// ============================================
// DB_RecipeProgram1 - SpinningCam Program
// Lines: 445
// Generated by SpinningCam
// ============================================

DATA_BLOCK "DB_RecipeProgram1"
{ S7_Optimized_Access := 'TRUE' }
VERSION : 0.1
NON_RETAIN
    VAR
        Header : "RecipeHeader";
        Lines : Array[0..999] of "RecipeLine";
    END_VAR
BEGIN
    // Header
    Header.Name := 'SpinningCam Program';
    Header.LineCount := 445;
    Header.Valid := TRUE;
    Header.PreScanned := FALSE;
    Header.MinX := 0.000;
    Header.MaxX := 118.345;
    Header.MinZ := -188.810;
    Header.MaxZ := 0.000;

    // Recipe Lines (445 total)
    Lines[0].X := 0.000; Lines[0].Z := 0.000; Lines[0].F := 0; Lines[0].CMD := 0; Lines[0].Param := 0; // G0 Rapid
    Lines[1].X := 0.000; Lines[1].Z := 0.000; Lines[1].F := 0; Lines[1].CMD := 0; Lines[1].Param := 0; // G0 Rapid
    Lines[2].X := 0.000; Lines[2].Z := 0.000; Lines[2].F := 0; Lines[2].CMD := 10; Lines[2].Param := 101; // Tool Change T101
    Lines[3].X := 0.000; Lines[3].Z := 0.000; Lines[3].F := 0; Lines[3].CMD := 20; Lines[3].Param := 20; // Spindle ON 200 RPM
    Lines[4].X := 34.600; Lines[4].Z := -28.936; Lines[4].F := 0; Lines[4].CMD := 0; Lines[4].Param := 0; // G0 Rapid
    Lines[5].X := 35.427; Lines[5].Z := -29.545; Lines[5].F := 300; Lines[5].CMD := 1; Lines[5].Param := 0; // G1 Linear
    Lines[6].X := 36.268; Lines[6].Z := -30.173; Lines[6].F := 300; Lines[6].CMD := 1; Lines[6].Param := 0; // G1 Linear
    Lines[7].X := 37.121; Lines[7].Z := -30.818; Lines[7].F := 300; Lines[7].CMD := 1; Lines[7].Param := 0; // G1 Linear
    Lines[8].X := 37.986; Lines[8].Z := -31.481; Lines[8].F := 300; Lines[8].CMD := 1; Lines[8].Param := 0; // G1 Linear
    Lines[9].X := 38.860; Lines[9].Z := -32.160; Lines[9].F := 300; Lines[9].CMD := 1; Lines[9].Param := 0; // G1 Linear
    Lines[10].X := 39.744; Lines[10].Z := -32.855; Lines[10].F := 300; Lines[10].CMD := 1; Lines[10].Param := 0; // G1 Linear
    Lines[11].X := 40.636; Lines[11].Z := -33.566; Lines[11].F := 300; Lines[11].CMD := 1; Lines[11].Param := 0; // G1 Linear
    Lines[12].X := 41.535; Lines[12].Z := -34.291; Lines[12].F := 300; Lines[12].CMD := 1; Lines[12].Param := 0; // G1 Linear
    Lines[13].X := 42.441; Lines[13].Z := -35.031; Lines[13].F := 300; Lines[13].CMD := 1; Lines[13].Param := 0; // G1 Linear
    Lines[14].X := 43.351; Lines[14].Z := -35.785; Lines[14].F := 300; Lines[14].CMD := 1; Lines[14].Param := 0; // G1 Linear
    Lines[15].X := 44.265; Lines[15].Z := -36.552; Lines[15].F := 300; Lines[15].CMD := 1; Lines[15].Param := 0; // G1 Linear
    Lines[16].X := 45.183; Lines[16].Z := -37.332; Lines[16].F := 300; Lines[16].CMD := 1; Lines[16].Param := 0; // G1 Linear
    Lines[17].X := 46.102; Lines[17].Z := -38.124; Lines[17].F := 300; Lines[17].CMD := 1; Lines[17].Param := 0; // G1 Linear
    Lines[18].X := 47.022; Lines[18].Z := -38.928; Lines[18].F := 300; Lines[18].CMD := 1; Lines[18].Param := 0; // G1 Linear
    Lines[19].X := 47.942; Lines[19].Z := -39.743; Lines[19].F := 300; Lines[19].CMD := 1; Lines[19].Param := 0; // G1 Linear
    Lines[20].X := 48.861; Lines[20].Z := -40.568; Lines[20].F := 300; Lines[20].CMD := 1; Lines[20].Param := 0; // G1 Linear
    Lines[21].X := 49.777; Lines[21].Z := -41.404; Lines[21].F := 300; Lines[21].CMD := 1; Lines[21].Param := 0; // G1 Linear
    Lines[22].X := 50.691; Lines[22].Z := -42.249; Lines[22].F := 300; Lines[22].CMD := 1; Lines[22].Param := 0; // G1 Linear
    Lines[23].X := 51.600; Lines[23].Z := -43.103; Lines[23].F := 300; Lines[23].CMD := 1; Lines[23].Param := 0; // G1 Linear
    Lines[24].X := 52.503; Lines[24].Z := -43.965; Lines[24].F := 300; Lines[24].CMD := 1; Lines[24].Param := 0; // G1 Linear
    Lines[25].X := 53.401; Lines[25].Z := -44.835; Lines[25].F := 300; Lines[25].CMD := 1; Lines[25].Param := 0; // G1 Linear
    Lines[26].X := 54.291; Lines[26].Z := -45.713; Lines[26].F := 300; Lines[26].CMD := 1; Lines[26].Param := 0; // G1 Linear
    Lines[27].X := 55.172; Lines[27].Z := -46.597; Lines[27].F := 300; Lines[27].CMD := 1; Lines[27].Param := 0; // G1 Linear
    Lines[28].X := 56.044; Lines[28].Z := -47.488; Lines[28].F := 300; Lines[28].CMD := 1; Lines[28].Param := 0; // G1 Linear
    Lines[29].X := 56.905; Lines[29].Z := -48.384; Lines[29].F := 300; Lines[29].CMD := 1; Lines[29].Param := 0; // G1 Linear
    Lines[30].X := 57.755; Lines[30].Z := -49.285; Lines[30].F := 300; Lines[30].CMD := 1; Lines[30].Param := 0; // G1 Linear
    Lines[31].X := 58.592; Lines[31].Z := -50.191; Lines[31].F := 300; Lines[31].CMD := 1; Lines[31].Param := 0; // G1 Linear
    Lines[32].X := 59.415; Lines[32].Z := -51.101; Lines[32].F := 300; Lines[32].CMD := 1; Lines[32].Param := 0; // G1 Linear
    Lines[33].X := 60.224; Lines[33].Z := -52.014; Lines[33].F := 300; Lines[33].CMD := 1; Lines[33].Param := 0; // G1 Linear
    Lines[34].X := 61.017; Lines[34].Z := -52.931; Lines[34].F := 300; Lines[34].CMD := 1; Lines[34].Param := 0; // G1 Linear
    Lines[35].X := 61.793; Lines[35].Z := -53.849; Lines[35].F := 300; Lines[35].CMD := 1; Lines[35].Param := 0; // G1 Linear
    Lines[36].X := 62.551; Lines[36].Z := -54.770; Lines[36].F := 300; Lines[36].CMD := 1; Lines[36].Param := 0; // G1 Linear
    Lines[37].X := 63.291; Lines[37].Z := -55.692; Lines[37].F := 300; Lines[37].CMD := 1; Lines[37].Param := 0; // G1 Linear
    Lines[38].X := 64.010; Lines[38].Z := -56.614; Lines[38].F := 300; Lines[38].CMD := 1; Lines[38].Param := 0; // G1 Linear
    Lines[39].X := 64.709; Lines[39].Z := -57.537; Lines[39].F := 300; Lines[39].CMD := 1; Lines[39].Param := 0; // G1 Linear
    Lines[40].X := 65.385; Lines[40].Z := -58.460; Lines[40].F := 300; Lines[40].CMD := 1; Lines[40].Param := 0; // G1 Linear
    Lines[41].X := 66.039; Lines[41].Z := -59.381; Lines[41].F := 300; Lines[41].CMD := 1; Lines[41].Param := 0; // G1 Linear
    Lines[42].X := 66.668; Lines[42].Z := -60.301; Lines[42].F := 300; Lines[42].CMD := 1; Lines[42].Param := 0; // G1 Linear
    Lines[43].X := 67.273; Lines[43].Z := -61.220; Lines[43].F := 300; Lines[43].CMD := 1; Lines[43].Param := 0; // G1 Linear
    Lines[44].X := 67.851; Lines[44].Z := -62.135; Lines[44].F := 300; Lines[44].CMD := 1; Lines[44].Param := 0; // G1 Linear
    Lines[45].X := 68.402; Lines[45].Z := -63.048; Lines[45].F := 300; Lines[45].CMD := 1; Lines[45].Param := 0; // G1 Linear
    Lines[46].X := 68.924; Lines[46].Z := -63.957; Lines[46].F := 300; Lines[46].CMD := 1; Lines[46].Param := 0; // G1 Linear
    Lines[47].X := 69.418; Lines[47].Z := -64.862; Lines[47].F := 300; Lines[47].CMD := 1; Lines[47].Param := 0; // G1 Linear
    Lines[48].X := 69.881; Lines[48].Z := -65.762; Lines[48].F := 300; Lines[48].CMD := 1; Lines[48].Param := 0; // G1 Linear
    Lines[49].X := 70.313; Lines[49].Z := -66.657; Lines[49].F := 300; Lines[49].CMD := 1; Lines[49].Param := 0; // G1 Linear
    Lines[50].X := 70.712; Lines[50].Z := -67.546; Lines[50].F := 300; Lines[50].CMD := 1; Lines[50].Param := 0; // G1 Linear
    Lines[51].X := 71.078; Lines[51].Z := -68.428; Lines[51].F := 300; Lines[51].CMD := 1; Lines[51].Param := 0; // G1 Linear
    Lines[52].X := 71.409; Lines[52].Z := -69.304; Lines[52].F := 300; Lines[52].CMD := 1; Lines[52].Param := 0; // G1 Linear
    Lines[53].X := 71.705; Lines[53].Z := -70.173; Lines[53].F := 300; Lines[53].CMD := 1; Lines[53].Param := 0; // G1 Linear
    Lines[54].X := 71.964; Lines[54].Z := -71.033; Lines[54].F := 300; Lines[54].CMD := 1; Lines[54].Param := 0; // G1 Linear
    Lines[55].X := 72.186; Lines[55].Z := -71.885; Lines[55].F := 300; Lines[55].CMD := 1; Lines[55].Param := 0; // G1 Linear
    Lines[56].X := 72.369; Lines[56].Z := -72.728; Lines[56].F := 300; Lines[56].CMD := 1; Lines[56].Param := 0; // G1 Linear
    Lines[57].X := 72.512; Lines[57].Z := -73.561; Lines[57].F := 300; Lines[57].CMD := 1; Lines[57].Param := 0; // G1 Linear
    Lines[58].X := 72.614; Lines[58].Z := -74.384; Lines[58].F := 300; Lines[58].CMD := 1; Lines[58].Param := 0; // G1 Linear
    Lines[59].X := 72.675; Lines[59].Z := -75.196; Lines[59].F := 300; Lines[59].CMD := 1; Lines[59].Param := 0; // G1 Linear
    Lines[60].X := 72.693; Lines[60].Z := -75.997; Lines[60].F := 300; Lines[60].CMD := 1; Lines[60].Param := 0; // G1 Linear
    Lines[61].X := 72.667; Lines[61].Z := -76.786; Lines[61].F := 300; Lines[61].CMD := 1; Lines[61].Param := 0; // G1 Linear
    Lines[62].X := 72.596; Lines[62].Z := -77.563; Lines[62].F := 300; Lines[62].CMD := 1; Lines[62].Param := 0; // G1 Linear
    Lines[63].X := 72.480; Lines[63].Z := -78.327; Lines[63].F := 300; Lines[63].CMD := 1; Lines[63].Param := 0; // G1 Linear
    Lines[64].X := 72.316; Lines[64].Z := -79.078; Lines[64].F := 300; Lines[64].CMD := 1; Lines[64].Param := 0; // G1 Linear
    Lines[65].X := 72.104; Lines[65].Z := -79.814; Lines[65].F := 300; Lines[65].CMD := 1; Lines[65].Param := 0; // G1 Linear
    Lines[66].X := 71.843; Lines[66].Z := -80.536; Lines[66].F := 300; Lines[66].CMD := 1; Lines[66].Param := 0; // G1 Linear
    Lines[67].X := 71.532; Lines[67].Z := -81.243; Lines[67].F := 300; Lines[67].CMD := 1; Lines[67].Param := 0; // G1 Linear
    Lines[68].X := 71.171; Lines[68].Z := -81.935; Lines[68].F := 300; Lines[68].CMD := 1; Lines[68].Param := 0; // G1 Linear
    Lines[69].X := 70.760; Lines[69].Z := -82.610; Lines[69].F := 300; Lines[69].CMD := 1; Lines[69].Param := 0; // G1 Linear
    Lines[70].X := 70.301; Lines[70].Z := -83.271; Lines[70].F := 300; Lines[70].CMD := 1; Lines[70].Param := 0; // G1 Linear
    Lines[71].X := 69.795; Lines[71].Z := -83.916; Lines[71].F := 300; Lines[71].CMD := 1; Lines[71].Param := 0; // G1 Linear
    Lines[72].X := 69.245; Lines[72].Z := -84.547; Lines[72].F := 300; Lines[72].CMD := 1; Lines[72].Param := 0; // G1 Linear
    Lines[73].X := 68.652; Lines[73].Z := -85.162; Lines[73].F := 300; Lines[73].CMD := 1; Lines[73].Param := 0; // G1 Linear
    Lines[74].X := 68.018; Lines[74].Z := -85.762; Lines[74].F := 300; Lines[74].CMD := 1; Lines[74].Param := 0; // G1 Linear
    Lines[75].X := 67.344; Lines[75].Z := -86.348; Lines[75].F := 300; Lines[75].CMD := 1; Lines[75].Param := 0; // G1 Linear
    Lines[76].X := 66.632; Lines[76].Z := -86.919; Lines[76].F := 300; Lines[76].CMD := 1; Lines[76].Param := 0; // G1 Linear
    Lines[77].X := 65.884; Lines[77].Z := -87.476; Lines[77].F := 300; Lines[77].CMD := 1; Lines[77].Param := 0; // G1 Linear
    Lines[78].X := 65.101; Lines[78].Z := -88.019; Lines[78].F := 300; Lines[78].CMD := 1; Lines[78].Param := 0; // G1 Linear
    Lines[79].X := 64.284; Lines[79].Z := -88.547; Lines[79].F := 300; Lines[79].CMD := 1; Lines[79].Param := 0; // G1 Linear
    Lines[80].X := 63.436; Lines[80].Z := -89.062; Lines[80].F := 300; Lines[80].CMD := 1; Lines[80].Param := 0; // G1 Linear
    Lines[81].X := 62.558; Lines[81].Z := -89.562; Lines[81].F := 300; Lines[81].CMD := 1; Lines[81].Param := 0; // G1 Linear
    Lines[82].X := 61.652; Lines[82].Z := -90.049; Lines[82].F := 300; Lines[82].CMD := 1; Lines[82].Param := 0; // G1 Linear
    Lines[83].X := 60.719; Lines[83].Z := -90.523; Lines[83].F := 300; Lines[83].CMD := 1; Lines[83].Param := 0; // G1 Linear
    Lines[84].X := 59.761; Lines[84].Z := -90.982; Lines[84].F := 300; Lines[84].CMD := 1; Lines[84].Param := 0; // G1 Linear
    Lines[85].X := 58.780; Lines[85].Z := -91.429; Lines[85].F := 300; Lines[85].CMD := 1; Lines[85].Param := 0; // G1 Linear
    Lines[86].X := 57.777; Lines[86].Z := -91.862; Lines[86].F := 300; Lines[86].CMD := 1; Lines[86].Param := 0; // G1 Linear
    Lines[87].X := 56.754; Lines[87].Z := -92.283; Lines[87].F := 300; Lines[87].CMD := 1; Lines[87].Param := 0; // G1 Linear
    Lines[88].X := 55.712; Lines[88].Z := -92.690; Lines[88].F := 300; Lines[88].CMD := 1; Lines[88].Param := 0; // G1 Linear
    Lines[89].X := 54.654; Lines[89].Z := -93.085; Lines[89].F := 300; Lines[89].CMD := 1; Lines[89].Param := 0; // G1 Linear
    Lines[90].X := 53.580; Lines[90].Z := -93.467; Lines[90].F := 300; Lines[90].CMD := 1; Lines[90].Param := 0; // G1 Linear
    Lines[91].X := 52.493; Lines[91].Z := -93.836; Lines[91].F := 300; Lines[91].CMD := 1; Lines[91].Param := 0; // G1 Linear
    Lines[92].X := 51.393; Lines[92].Z := -94.193; Lines[92].F := 300; Lines[92].CMD := 1; Lines[92].Param := 0; // G1 Linear
    Lines[93].X := 50.284; Lines[93].Z := -94.538; Lines[93].F := 300; Lines[93].CMD := 1; Lines[93].Param := 0; // G1 Linear
    Lines[94].X := 49.165; Lines[94].Z := -94.871; Lines[94].F := 300; Lines[94].CMD := 1; Lines[94].Param := 0; // G1 Linear
    Lines[95].X := 48.040; Lines[95].Z := -95.192; Lines[95].F := 300; Lines[95].CMD := 1; Lines[95].Param := 0; // G1 Linear
    Lines[96].X := 46.909; Lines[96].Z := -95.501; Lines[96].F := 300; Lines[96].CMD := 1; Lines[96].Param := 0; // G1 Linear
    Lines[97].X := 45.775; Lines[97].Z := -95.798; Lines[97].F := 300; Lines[97].CMD := 1; Lines[97].Param := 0; // G1 Linear
    Lines[98].X := 44.638; Lines[98].Z := -96.084; Lines[98].F := 300; Lines[98].CMD := 1; Lines[98].Param := 0; // G1 Linear
    Lines[99].X := 43.501; Lines[99].Z := -96.358; Lines[99].F := 300; Lines[99].CMD := 1; Lines[99].Param := 0; // G1 Linear
    Lines[100].X := 42.364; Lines[100].Z := -96.621; Lines[100].F := 300; Lines[100].CMD := 1; Lines[100].Param := 0; // G1 Linear
    Lines[101].X := 41.231; Lines[101].Z := -96.873; Lines[101].F := 300; Lines[101].CMD := 1; Lines[101].Param := 0; // G1 Linear
    Lines[102].X := 40.102; Lines[102].Z := -97.114; Lines[102].F := 300; Lines[102].CMD := 1; Lines[102].Param := 0; // G1 Linear
    Lines[103].X := 38.979; Lines[103].Z := -97.344; Lines[103].F := 300; Lines[103].CMD := 1; Lines[103].Param := 0; // G1 Linear
    Lines[104].X := 37.863; Lines[104].Z := -97.564; Lines[104].F := 300; Lines[104].CMD := 1; Lines[104].Param := 0; // G1 Linear
    Lines[105].X := 36.757; Lines[105].Z := -97.772; Lines[105].F := 300; Lines[105].CMD := 1; Lines[105].Param := 0; // G1 Linear
    Lines[106].X := 35.662; Lines[106].Z := -97.971; Lines[106].F := 300; Lines[106].CMD := 1; Lines[106].Param := 0; // G1 Linear
    Lines[107].X := 34.579; Lines[107].Z := -98.159; Lines[107].F := 300; Lines[107].CMD := 1; Lines[107].Param := 0; // G1 Linear
    Lines[108].X := 33.511; Lines[108].Z := -98.337; Lines[108].F := 300; Lines[108].CMD := 1; Lines[108].Param := 0; // G1 Linear
    Lines[109].X := 32.458; Lines[109].Z := -98.504; Lines[109].F := 300; Lines[109].CMD := 1; Lines[109].Param := 0; // G1 Linear
    Lines[110].X := 31.422; Lines[110].Z := -98.662; Lines[110].F := 300; Lines[110].CMD := 1; Lines[110].Param := 0; // G1 Linear
    Lines[111].X := 30.406; Lines[111].Z := -98.810; Lines[111].F := 300; Lines[111].CMD := 1; Lines[111].Param := 0; // G1 Linear
    Lines[112].X := 10.406; Lines[112].Z := -78.810; Lines[112].F := 0; Lines[112].CMD := 0; Lines[112].Param := 0; // G0 Rapid
    Lines[113].X := 49.600; Lines[113].Z := -58.936; Lines[113].F := 0; Lines[113].CMD := 0; Lines[113].Param := 0; // G0 Rapid
    Lines[114].X := 50.427; Lines[114].Z := -59.545; Lines[114].F := 300; Lines[114].CMD := 1; Lines[114].Param := 0; // G1 Linear
    Lines[115].X := 51.268; Lines[115].Z := -60.173; Lines[115].F := 300; Lines[115].CMD := 1; Lines[115].Param := 0; // G1 Linear
    Lines[116].X := 52.121; Lines[116].Z := -60.818; Lines[116].F := 300; Lines[116].CMD := 1; Lines[116].Param := 0; // G1 Linear
    Lines[117].X := 52.986; Lines[117].Z := -61.481; Lines[117].F := 300; Lines[117].CMD := 1; Lines[117].Param := 0; // G1 Linear
    Lines[118].X := 53.860; Lines[118].Z := -62.160; Lines[118].F := 300; Lines[118].CMD := 1; Lines[118].Param := 0; // G1 Linear
    Lines[119].X := 54.744; Lines[119].Z := -62.855; Lines[119].F := 300; Lines[119].CMD := 1; Lines[119].Param := 0; // G1 Linear
    Lines[120].X := 55.636; Lines[120].Z := -63.566; Lines[120].F := 300; Lines[120].CMD := 1; Lines[120].Param := 0; // G1 Linear
    Lines[121].X := 56.535; Lines[121].Z := -64.291; Lines[121].F := 300; Lines[121].CMD := 1; Lines[121].Param := 0; // G1 Linear
    Lines[122].X := 57.441; Lines[122].Z := -65.031; Lines[122].F := 300; Lines[122].CMD := 1; Lines[122].Param := 0; // G1 Linear
    Lines[123].X := 58.351; Lines[123].Z := -65.785; Lines[123].F := 300; Lines[123].CMD := 1; Lines[123].Param := 0; // G1 Linear
    Lines[124].X := 59.265; Lines[124].Z := -66.552; Lines[124].F := 300; Lines[124].CMD := 1; Lines[124].Param := 0; // G1 Linear
    Lines[125].X := 60.183; Lines[125].Z := -67.332; Lines[125].F := 300; Lines[125].CMD := 1; Lines[125].Param := 0; // G1 Linear
    Lines[126].X := 61.102; Lines[126].Z := -68.124; Lines[126].F := 300; Lines[126].CMD := 1; Lines[126].Param := 0; // G1 Linear
    Lines[127].X := 62.022; Lines[127].Z := -68.928; Lines[127].F := 300; Lines[127].CMD := 1; Lines[127].Param := 0; // G1 Linear
    Lines[128].X := 62.942; Lines[128].Z := -69.743; Lines[128].F := 300; Lines[128].CMD := 1; Lines[128].Param := 0; // G1 Linear
    Lines[129].X := 63.861; Lines[129].Z := -70.568; Lines[129].F := 300; Lines[129].CMD := 1; Lines[129].Param := 0; // G1 Linear
    Lines[130].X := 64.777; Lines[130].Z := -71.404; Lines[130].F := 300; Lines[130].CMD := 1; Lines[130].Param := 0; // G1 Linear
    Lines[131].X := 65.691; Lines[131].Z := -72.249; Lines[131].F := 300; Lines[131].CMD := 1; Lines[131].Param := 0; // G1 Linear
    Lines[132].X := 66.600; Lines[132].Z := -73.103; Lines[132].F := 300; Lines[132].CMD := 1; Lines[132].Param := 0; // G1 Linear
    Lines[133].X := 67.503; Lines[133].Z := -73.965; Lines[133].F := 300; Lines[133].CMD := 1; Lines[133].Param := 0; // G1 Linear
    Lines[134].X := 68.401; Lines[134].Z := -74.835; Lines[134].F := 300; Lines[134].CMD := 1; Lines[134].Param := 0; // G1 Linear
    Lines[135].X := 69.291; Lines[135].Z := -75.713; Lines[135].F := 300; Lines[135].CMD := 1; Lines[135].Param := 0; // G1 Linear
    Lines[136].X := 70.172; Lines[136].Z := -76.597; Lines[136].F := 300; Lines[136].CMD := 1; Lines[136].Param := 0; // G1 Linear
    Lines[137].X := 71.044; Lines[137].Z := -77.488; Lines[137].F := 300; Lines[137].CMD := 1; Lines[137].Param := 0; // G1 Linear
    Lines[138].X := 71.905; Lines[138].Z := -78.384; Lines[138].F := 300; Lines[138].CMD := 1; Lines[138].Param := 0; // G1 Linear
    Lines[139].X := 72.755; Lines[139].Z := -79.285; Lines[139].F := 300; Lines[139].CMD := 1; Lines[139].Param := 0; // G1 Linear
    Lines[140].X := 73.592; Lines[140].Z := -80.191; Lines[140].F := 300; Lines[140].CMD := 1; Lines[140].Param := 0; // G1 Linear
    Lines[141].X := 74.415; Lines[141].Z := -81.101; Lines[141].F := 300; Lines[141].CMD := 1; Lines[141].Param := 0; // G1 Linear
    Lines[142].X := 75.224; Lines[142].Z := -82.014; Lines[142].F := 300; Lines[142].CMD := 1; Lines[142].Param := 0; // G1 Linear
    Lines[143].X := 76.017; Lines[143].Z := -82.931; Lines[143].F := 300; Lines[143].CMD := 1; Lines[143].Param := 0; // G1 Linear
    Lines[144].X := 76.793; Lines[144].Z := -83.849; Lines[144].F := 300; Lines[144].CMD := 1; Lines[144].Param := 0; // G1 Linear
    Lines[145].X := 77.551; Lines[145].Z := -84.770; Lines[145].F := 300; Lines[145].CMD := 1; Lines[145].Param := 0; // G1 Linear
    Lines[146].X := 78.291; Lines[146].Z := -85.692; Lines[146].F := 300; Lines[146].CMD := 1; Lines[146].Param := 0; // G1 Linear
    Lines[147].X := 79.010; Lines[147].Z := -86.614; Lines[147].F := 300; Lines[147].CMD := 1; Lines[147].Param := 0; // G1 Linear
    Lines[148].X := 79.709; Lines[148].Z := -87.537; Lines[148].F := 300; Lines[148].CMD := 1; Lines[148].Param := 0; // G1 Linear
    Lines[149].X := 80.385; Lines[149].Z := -88.460; Lines[149].F := 300; Lines[149].CMD := 1; Lines[149].Param := 0; // G1 Linear
    Lines[150].X := 81.039; Lines[150].Z := -89.381; Lines[150].F := 300; Lines[150].CMD := 1; Lines[150].Param := 0; // G1 Linear
    Lines[151].X := 81.668; Lines[151].Z := -90.301; Lines[151].F := 300; Lines[151].CMD := 1; Lines[151].Param := 0; // G1 Linear
    Lines[152].X := 82.273; Lines[152].Z := -91.220; Lines[152].F := 300; Lines[152].CMD := 1; Lines[152].Param := 0; // G1 Linear
    Lines[153].X := 82.851; Lines[153].Z := -92.135; Lines[153].F := 300; Lines[153].CMD := 1; Lines[153].Param := 0; // G1 Linear
    Lines[154].X := 83.402; Lines[154].Z := -93.048; Lines[154].F := 300; Lines[154].CMD := 1; Lines[154].Param := 0; // G1 Linear
    Lines[155].X := 83.924; Lines[155].Z := -93.957; Lines[155].F := 300; Lines[155].CMD := 1; Lines[155].Param := 0; // G1 Linear
    Lines[156].X := 84.418; Lines[156].Z := -94.862; Lines[156].F := 300; Lines[156].CMD := 1; Lines[156].Param := 0; // G1 Linear
    Lines[157].X := 84.881; Lines[157].Z := -95.762; Lines[157].F := 300; Lines[157].CMD := 1; Lines[157].Param := 0; // G1 Linear
    Lines[158].X := 85.313; Lines[158].Z := -96.657; Lines[158].F := 300; Lines[158].CMD := 1; Lines[158].Param := 0; // G1 Linear
    Lines[159].X := 85.712; Lines[159].Z := -97.546; Lines[159].F := 300; Lines[159].CMD := 1; Lines[159].Param := 0; // G1 Linear
    Lines[160].X := 86.078; Lines[160].Z := -98.428; Lines[160].F := 300; Lines[160].CMD := 1; Lines[160].Param := 0; // G1 Linear
    Lines[161].X := 86.409; Lines[161].Z := -99.304; Lines[161].F := 300; Lines[161].CMD := 1; Lines[161].Param := 0; // G1 Linear
    Lines[162].X := 86.705; Lines[162].Z := -100.173; Lines[162].F := 300; Lines[162].CMD := 1; Lines[162].Param := 0; // G1 Linear
    Lines[163].X := 86.964; Lines[163].Z := -101.033; Lines[163].F := 300; Lines[163].CMD := 1; Lines[163].Param := 0; // G1 Linear
    Lines[164].X := 87.186; Lines[164].Z := -101.885; Lines[164].F := 300; Lines[164].CMD := 1; Lines[164].Param := 0; // G1 Linear
    Lines[165].X := 87.369; Lines[165].Z := -102.728; Lines[165].F := 300; Lines[165].CMD := 1; Lines[165].Param := 0; // G1 Linear
    Lines[166].X := 87.512; Lines[166].Z := -103.561; Lines[166].F := 300; Lines[166].CMD := 1; Lines[166].Param := 0; // G1 Linear
    Lines[167].X := 87.614; Lines[167].Z := -104.384; Lines[167].F := 300; Lines[167].CMD := 1; Lines[167].Param := 0; // G1 Linear
    Lines[168].X := 87.675; Lines[168].Z := -105.196; Lines[168].F := 300; Lines[168].CMD := 1; Lines[168].Param := 0; // G1 Linear
    Lines[169].X := 87.693; Lines[169].Z := -105.997; Lines[169].F := 300; Lines[169].CMD := 1; Lines[169].Param := 0; // G1 Linear
    Lines[170].X := 87.667; Lines[170].Z := -106.786; Lines[170].F := 300; Lines[170].CMD := 1; Lines[170].Param := 0; // G1 Linear
    Lines[171].X := 87.596; Lines[171].Z := -107.563; Lines[171].F := 300; Lines[171].CMD := 1; Lines[171].Param := 0; // G1 Linear
    Lines[172].X := 87.480; Lines[172].Z := -108.327; Lines[172].F := 300; Lines[172].CMD := 1; Lines[172].Param := 0; // G1 Linear
    Lines[173].X := 87.316; Lines[173].Z := -109.078; Lines[173].F := 300; Lines[173].CMD := 1; Lines[173].Param := 0; // G1 Linear
    Lines[174].X := 87.104; Lines[174].Z := -109.814; Lines[174].F := 300; Lines[174].CMD := 1; Lines[174].Param := 0; // G1 Linear
    Lines[175].X := 86.843; Lines[175].Z := -110.536; Lines[175].F := 300; Lines[175].CMD := 1; Lines[175].Param := 0; // G1 Linear
    Lines[176].X := 86.532; Lines[176].Z := -111.243; Lines[176].F := 300; Lines[176].CMD := 1; Lines[176].Param := 0; // G1 Linear
    Lines[177].X := 86.171; Lines[177].Z := -111.935; Lines[177].F := 300; Lines[177].CMD := 1; Lines[177].Param := 0; // G1 Linear
    Lines[178].X := 85.760; Lines[178].Z := -112.610; Lines[178].F := 300; Lines[178].CMD := 1; Lines[178].Param := 0; // G1 Linear
    Lines[179].X := 85.301; Lines[179].Z := -113.271; Lines[179].F := 300; Lines[179].CMD := 1; Lines[179].Param := 0; // G1 Linear
    Lines[180].X := 84.795; Lines[180].Z := -113.916; Lines[180].F := 300; Lines[180].CMD := 1; Lines[180].Param := 0; // G1 Linear
    Lines[181].X := 84.245; Lines[181].Z := -114.547; Lines[181].F := 300; Lines[181].CMD := 1; Lines[181].Param := 0; // G1 Linear
    Lines[182].X := 83.652; Lines[182].Z := -115.162; Lines[182].F := 300; Lines[182].CMD := 1; Lines[182].Param := 0; // G1 Linear
    Lines[183].X := 83.018; Lines[183].Z := -115.762; Lines[183].F := 300; Lines[183].CMD := 1; Lines[183].Param := 0; // G1 Linear
    Lines[184].X := 82.344; Lines[184].Z := -116.348; Lines[184].F := 300; Lines[184].CMD := 1; Lines[184].Param := 0; // G1 Linear
    Lines[185].X := 81.632; Lines[185].Z := -116.919; Lines[185].F := 300; Lines[185].CMD := 1; Lines[185].Param := 0; // G1 Linear
    Lines[186].X := 80.884; Lines[186].Z := -117.476; Lines[186].F := 300; Lines[186].CMD := 1; Lines[186].Param := 0; // G1 Linear
    Lines[187].X := 80.101; Lines[187].Z := -118.019; Lines[187].F := 300; Lines[187].CMD := 1; Lines[187].Param := 0; // G1 Linear
    Lines[188].X := 79.284; Lines[188].Z := -118.547; Lines[188].F := 300; Lines[188].CMD := 1; Lines[188].Param := 0; // G1 Linear
    Lines[189].X := 78.436; Lines[189].Z := -119.062; Lines[189].F := 300; Lines[189].CMD := 1; Lines[189].Param := 0; // G1 Linear
    Lines[190].X := 77.558; Lines[190].Z := -119.562; Lines[190].F := 300; Lines[190].CMD := 1; Lines[190].Param := 0; // G1 Linear
    Lines[191].X := 76.652; Lines[191].Z := -120.049; Lines[191].F := 300; Lines[191].CMD := 1; Lines[191].Param := 0; // G1 Linear
    Lines[192].X := 75.719; Lines[192].Z := -120.523; Lines[192].F := 300; Lines[192].CMD := 1; Lines[192].Param := 0; // G1 Linear
    Lines[193].X := 74.761; Lines[193].Z := -120.982; Lines[193].F := 300; Lines[193].CMD := 1; Lines[193].Param := 0; // G1 Linear
    Lines[194].X := 73.780; Lines[194].Z := -121.429; Lines[194].F := 300; Lines[194].CMD := 1; Lines[194].Param := 0; // G1 Linear
    Lines[195].X := 72.777; Lines[195].Z := -121.862; Lines[195].F := 300; Lines[195].CMD := 1; Lines[195].Param := 0; // G1 Linear
    Lines[196].X := 71.754; Lines[196].Z := -122.283; Lines[196].F := 300; Lines[196].CMD := 1; Lines[196].Param := 0; // G1 Linear
    Lines[197].X := 70.712; Lines[197].Z := -122.690; Lines[197].F := 300; Lines[197].CMD := 1; Lines[197].Param := 0; // G1 Linear
    Lines[198].X := 69.654; Lines[198].Z := -123.085; Lines[198].F := 300; Lines[198].CMD := 1; Lines[198].Param := 0; // G1 Linear
    Lines[199].X := 68.580; Lines[199].Z := -123.467; Lines[199].F := 300; Lines[199].CMD := 1; Lines[199].Param := 0; // G1 Linear
    Lines[200].X := 67.493; Lines[200].Z := -123.836; Lines[200].F := 300; Lines[200].CMD := 1; Lines[200].Param := 0; // G1 Linear
    Lines[201].X := 66.393; Lines[201].Z := -124.193; Lines[201].F := 300; Lines[201].CMD := 1; Lines[201].Param := 0; // G1 Linear
    Lines[202].X := 65.284; Lines[202].Z := -124.538; Lines[202].F := 300; Lines[202].CMD := 1; Lines[202].Param := 0; // G1 Linear
    Lines[203].X := 64.165; Lines[203].Z := -124.871; Lines[203].F := 300; Lines[203].CMD := 1; Lines[203].Param := 0; // G1 Linear
    Lines[204].X := 63.040; Lines[204].Z := -125.192; Lines[204].F := 300; Lines[204].CMD := 1; Lines[204].Param := 0; // G1 Linear
    Lines[205].X := 61.909; Lines[205].Z := -125.501; Lines[205].F := 300; Lines[205].CMD := 1; Lines[205].Param := 0; // G1 Linear
    Lines[206].X := 60.775; Lines[206].Z := -125.798; Lines[206].F := 300; Lines[206].CMD := 1; Lines[206].Param := 0; // G1 Linear
    Lines[207].X := 59.638; Lines[207].Z := -126.084; Lines[207].F := 300; Lines[207].CMD := 1; Lines[207].Param := 0; // G1 Linear
    Lines[208].X := 58.501; Lines[208].Z := -126.358; Lines[208].F := 300; Lines[208].CMD := 1; Lines[208].Param := 0; // G1 Linear
    Lines[209].X := 57.364; Lines[209].Z := -126.621; Lines[209].F := 300; Lines[209].CMD := 1; Lines[209].Param := 0; // G1 Linear
    Lines[210].X := 56.231; Lines[210].Z := -126.873; Lines[210].F := 300; Lines[210].CMD := 1; Lines[210].Param := 0; // G1 Linear
    Lines[211].X := 55.102; Lines[211].Z := -127.114; Lines[211].F := 300; Lines[211].CMD := 1; Lines[211].Param := 0; // G1 Linear
    Lines[212].X := 53.979; Lines[212].Z := -127.344; Lines[212].F := 300; Lines[212].CMD := 1; Lines[212].Param := 0; // G1 Linear
    Lines[213].X := 52.863; Lines[213].Z := -127.564; Lines[213].F := 300; Lines[213].CMD := 1; Lines[213].Param := 0; // G1 Linear
    Lines[214].X := 51.757; Lines[214].Z := -127.772; Lines[214].F := 300; Lines[214].CMD := 1; Lines[214].Param := 0; // G1 Linear
    Lines[215].X := 50.662; Lines[215].Z := -127.971; Lines[215].F := 300; Lines[215].CMD := 1; Lines[215].Param := 0; // G1 Linear
    Lines[216].X := 49.579; Lines[216].Z := -128.159; Lines[216].F := 300; Lines[216].CMD := 1; Lines[216].Param := 0; // G1 Linear
    Lines[217].X := 48.511; Lines[217].Z := -128.337; Lines[217].F := 300; Lines[217].CMD := 1; Lines[217].Param := 0; // G1 Linear
    Lines[218].X := 47.458; Lines[218].Z := -128.504; Lines[218].F := 300; Lines[218].CMD := 1; Lines[218].Param := 0; // G1 Linear
    Lines[219].X := 46.422; Lines[219].Z := -128.662; Lines[219].F := 300; Lines[219].CMD := 1; Lines[219].Param := 0; // G1 Linear
    Lines[220].X := 45.406; Lines[220].Z := -128.810; Lines[220].F := 300; Lines[220].CMD := 1; Lines[220].Param := 0; // G1 Linear
    Lines[221].X := 25.406; Lines[221].Z := -108.810; Lines[221].F := 0; Lines[221].CMD := 0; Lines[221].Param := 0; // G0 Rapid
    Lines[222].X := 64.600; Lines[222].Z := -88.936; Lines[222].F := 0; Lines[222].CMD := 0; Lines[222].Param := 0; // G0 Rapid
    Lines[223].X := 65.427; Lines[223].Z := -89.545; Lines[223].F := 300; Lines[223].CMD := 1; Lines[223].Param := 0; // G1 Linear
    Lines[224].X := 66.268; Lines[224].Z := -90.173; Lines[224].F := 300; Lines[224].CMD := 1; Lines[224].Param := 0; // G1 Linear
    Lines[225].X := 67.121; Lines[225].Z := -90.818; Lines[225].F := 300; Lines[225].CMD := 1; Lines[225].Param := 0; // G1 Linear
    Lines[226].X := 67.986; Lines[226].Z := -91.481; Lines[226].F := 300; Lines[226].CMD := 1; Lines[226].Param := 0; // G1 Linear
    Lines[227].X := 68.860; Lines[227].Z := -92.160; Lines[227].F := 300; Lines[227].CMD := 1; Lines[227].Param := 0; // G1 Linear
    Lines[228].X := 69.744; Lines[228].Z := -92.855; Lines[228].F := 300; Lines[228].CMD := 1; Lines[228].Param := 0; // G1 Linear
    Lines[229].X := 70.636; Lines[229].Z := -93.566; Lines[229].F := 300; Lines[229].CMD := 1; Lines[229].Param := 0; // G1 Linear
    Lines[230].X := 71.535; Lines[230].Z := -94.291; Lines[230].F := 300; Lines[230].CMD := 1; Lines[230].Param := 0; // G1 Linear
    Lines[231].X := 72.441; Lines[231].Z := -95.031; Lines[231].F := 300; Lines[231].CMD := 1; Lines[231].Param := 0; // G1 Linear
    Lines[232].X := 73.351; Lines[232].Z := -95.785; Lines[232].F := 300; Lines[232].CMD := 1; Lines[232].Param := 0; // G1 Linear
    Lines[233].X := 74.265; Lines[233].Z := -96.552; Lines[233].F := 300; Lines[233].CMD := 1; Lines[233].Param := 0; // G1 Linear
    Lines[234].X := 75.183; Lines[234].Z := -97.332; Lines[234].F := 300; Lines[234].CMD := 1; Lines[234].Param := 0; // G1 Linear
    Lines[235].X := 76.102; Lines[235].Z := -98.124; Lines[235].F := 300; Lines[235].CMD := 1; Lines[235].Param := 0; // G1 Linear
    Lines[236].X := 77.022; Lines[236].Z := -98.928; Lines[236].F := 300; Lines[236].CMD := 1; Lines[236].Param := 0; // G1 Linear
    Lines[237].X := 77.942; Lines[237].Z := -99.743; Lines[237].F := 300; Lines[237].CMD := 1; Lines[237].Param := 0; // G1 Linear
    Lines[238].X := 78.861; Lines[238].Z := -100.568; Lines[238].F := 300; Lines[238].CMD := 1; Lines[238].Param := 0; // G1 Linear
    Lines[239].X := 79.777; Lines[239].Z := -101.404; Lines[239].F := 300; Lines[239].CMD := 1; Lines[239].Param := 0; // G1 Linear
    Lines[240].X := 80.691; Lines[240].Z := -102.249; Lines[240].F := 300; Lines[240].CMD := 1; Lines[240].Param := 0; // G1 Linear
    Lines[241].X := 81.600; Lines[241].Z := -103.103; Lines[241].F := 300; Lines[241].CMD := 1; Lines[241].Param := 0; // G1 Linear
    Lines[242].X := 82.503; Lines[242].Z := -103.965; Lines[242].F := 300; Lines[242].CMD := 1; Lines[242].Param := 0; // G1 Linear
    Lines[243].X := 83.401; Lines[243].Z := -104.835; Lines[243].F := 300; Lines[243].CMD := 1; Lines[243].Param := 0; // G1 Linear
    Lines[244].X := 84.291; Lines[244].Z := -105.713; Lines[244].F := 300; Lines[244].CMD := 1; Lines[244].Param := 0; // G1 Linear
    Lines[245].X := 85.172; Lines[245].Z := -106.597; Lines[245].F := 300; Lines[245].CMD := 1; Lines[245].Param := 0; // G1 Linear
    Lines[246].X := 86.044; Lines[246].Z := -107.488; Lines[246].F := 300; Lines[246].CMD := 1; Lines[246].Param := 0; // G1 Linear
    Lines[247].X := 86.905; Lines[247].Z := -108.384; Lines[247].F := 300; Lines[247].CMD := 1; Lines[247].Param := 0; // G1 Linear
    Lines[248].X := 87.755; Lines[248].Z := -109.285; Lines[248].F := 300; Lines[248].CMD := 1; Lines[248].Param := 0; // G1 Linear
    Lines[249].X := 88.592; Lines[249].Z := -110.191; Lines[249].F := 300; Lines[249].CMD := 1; Lines[249].Param := 0; // G1 Linear
    Lines[250].X := 89.415; Lines[250].Z := -111.101; Lines[250].F := 300; Lines[250].CMD := 1; Lines[250].Param := 0; // G1 Linear
    Lines[251].X := 90.224; Lines[251].Z := -112.014; Lines[251].F := 300; Lines[251].CMD := 1; Lines[251].Param := 0; // G1 Linear
    Lines[252].X := 91.017; Lines[252].Z := -112.931; Lines[252].F := 300; Lines[252].CMD := 1; Lines[252].Param := 0; // G1 Linear
    Lines[253].X := 91.793; Lines[253].Z := -113.849; Lines[253].F := 300; Lines[253].CMD := 1; Lines[253].Param := 0; // G1 Linear
    Lines[254].X := 92.551; Lines[254].Z := -114.770; Lines[254].F := 300; Lines[254].CMD := 1; Lines[254].Param := 0; // G1 Linear
    Lines[255].X := 93.291; Lines[255].Z := -115.692; Lines[255].F := 300; Lines[255].CMD := 1; Lines[255].Param := 0; // G1 Linear
    Lines[256].X := 94.010; Lines[256].Z := -116.614; Lines[256].F := 300; Lines[256].CMD := 1; Lines[256].Param := 0; // G1 Linear
    Lines[257].X := 94.709; Lines[257].Z := -117.537; Lines[257].F := 300; Lines[257].CMD := 1; Lines[257].Param := 0; // G1 Linear
    Lines[258].X := 95.385; Lines[258].Z := -118.460; Lines[258].F := 300; Lines[258].CMD := 1; Lines[258].Param := 0; // G1 Linear
    Lines[259].X := 96.039; Lines[259].Z := -119.381; Lines[259].F := 300; Lines[259].CMD := 1; Lines[259].Param := 0; // G1 Linear
    Lines[260].X := 96.668; Lines[260].Z := -120.301; Lines[260].F := 300; Lines[260].CMD := 1; Lines[260].Param := 0; // G1 Linear
    Lines[261].X := 97.273; Lines[261].Z := -121.220; Lines[261].F := 300; Lines[261].CMD := 1; Lines[261].Param := 0; // G1 Linear
    Lines[262].X := 97.851; Lines[262].Z := -122.135; Lines[262].F := 300; Lines[262].CMD := 1; Lines[262].Param := 0; // G1 Linear
    Lines[263].X := 98.402; Lines[263].Z := -123.048; Lines[263].F := 300; Lines[263].CMD := 1; Lines[263].Param := 0; // G1 Linear
    Lines[264].X := 98.924; Lines[264].Z := -123.957; Lines[264].F := 300; Lines[264].CMD := 1; Lines[264].Param := 0; // G1 Linear
    Lines[265].X := 99.418; Lines[265].Z := -124.862; Lines[265].F := 300; Lines[265].CMD := 1; Lines[265].Param := 0; // G1 Linear
    Lines[266].X := 99.881; Lines[266].Z := -125.762; Lines[266].F := 300; Lines[266].CMD := 1; Lines[266].Param := 0; // G1 Linear
    Lines[267].X := 100.313; Lines[267].Z := -126.657; Lines[267].F := 300; Lines[267].CMD := 1; Lines[267].Param := 0; // G1 Linear
    Lines[268].X := 100.712; Lines[268].Z := -127.546; Lines[268].F := 300; Lines[268].CMD := 1; Lines[268].Param := 0; // G1 Linear
    Lines[269].X := 101.078; Lines[269].Z := -128.428; Lines[269].F := 300; Lines[269].CMD := 1; Lines[269].Param := 0; // G1 Linear
    Lines[270].X := 101.409; Lines[270].Z := -129.304; Lines[270].F := 300; Lines[270].CMD := 1; Lines[270].Param := 0; // G1 Linear
    Lines[271].X := 101.705; Lines[271].Z := -130.173; Lines[271].F := 300; Lines[271].CMD := 1; Lines[271].Param := 0; // G1 Linear
    Lines[272].X := 101.964; Lines[272].Z := -131.033; Lines[272].F := 300; Lines[272].CMD := 1; Lines[272].Param := 0; // G1 Linear
    Lines[273].X := 102.186; Lines[273].Z := -131.885; Lines[273].F := 300; Lines[273].CMD := 1; Lines[273].Param := 0; // G1 Linear
    Lines[274].X := 102.369; Lines[274].Z := -132.728; Lines[274].F := 300; Lines[274].CMD := 1; Lines[274].Param := 0; // G1 Linear
    Lines[275].X := 102.512; Lines[275].Z := -133.561; Lines[275].F := 300; Lines[275].CMD := 1; Lines[275].Param := 0; // G1 Linear
    Lines[276].X := 102.614; Lines[276].Z := -134.384; Lines[276].F := 300; Lines[276].CMD := 1; Lines[276].Param := 0; // G1 Linear
    Lines[277].X := 102.675; Lines[277].Z := -135.196; Lines[277].F := 300; Lines[277].CMD := 1; Lines[277].Param := 0; // G1 Linear
    Lines[278].X := 102.693; Lines[278].Z := -135.997; Lines[278].F := 300; Lines[278].CMD := 1; Lines[278].Param := 0; // G1 Linear
    Lines[279].X := 102.667; Lines[279].Z := -136.786; Lines[279].F := 300; Lines[279].CMD := 1; Lines[279].Param := 0; // G1 Linear
    Lines[280].X := 102.596; Lines[280].Z := -137.563; Lines[280].F := 300; Lines[280].CMD := 1; Lines[280].Param := 0; // G1 Linear
    Lines[281].X := 102.480; Lines[281].Z := -138.327; Lines[281].F := 300; Lines[281].CMD := 1; Lines[281].Param := 0; // G1 Linear
    Lines[282].X := 102.316; Lines[282].Z := -139.078; Lines[282].F := 300; Lines[282].CMD := 1; Lines[282].Param := 0; // G1 Linear
    Lines[283].X := 102.104; Lines[283].Z := -139.814; Lines[283].F := 300; Lines[283].CMD := 1; Lines[283].Param := 0; // G1 Linear
    Lines[284].X := 101.843; Lines[284].Z := -140.536; Lines[284].F := 300; Lines[284].CMD := 1; Lines[284].Param := 0; // G1 Linear
    Lines[285].X := 101.532; Lines[285].Z := -141.243; Lines[285].F := 300; Lines[285].CMD := 1; Lines[285].Param := 0; // G1 Linear
    Lines[286].X := 101.171; Lines[286].Z := -141.935; Lines[286].F := 300; Lines[286].CMD := 1; Lines[286].Param := 0; // G1 Linear
    Lines[287].X := 100.760; Lines[287].Z := -142.610; Lines[287].F := 300; Lines[287].CMD := 1; Lines[287].Param := 0; // G1 Linear
    Lines[288].X := 100.301; Lines[288].Z := -143.271; Lines[288].F := 300; Lines[288].CMD := 1; Lines[288].Param := 0; // G1 Linear
    Lines[289].X := 99.795; Lines[289].Z := -143.916; Lines[289].F := 300; Lines[289].CMD := 1; Lines[289].Param := 0; // G1 Linear
    Lines[290].X := 99.245; Lines[290].Z := -144.547; Lines[290].F := 300; Lines[290].CMD := 1; Lines[290].Param := 0; // G1 Linear
    Lines[291].X := 98.652; Lines[291].Z := -145.162; Lines[291].F := 300; Lines[291].CMD := 1; Lines[291].Param := 0; // G1 Linear
    Lines[292].X := 98.018; Lines[292].Z := -145.762; Lines[292].F := 300; Lines[292].CMD := 1; Lines[292].Param := 0; // G1 Linear
    Lines[293].X := 97.344; Lines[293].Z := -146.348; Lines[293].F := 300; Lines[293].CMD := 1; Lines[293].Param := 0; // G1 Linear
    Lines[294].X := 96.632; Lines[294].Z := -146.919; Lines[294].F := 300; Lines[294].CMD := 1; Lines[294].Param := 0; // G1 Linear
    Lines[295].X := 95.884; Lines[295].Z := -147.476; Lines[295].F := 300; Lines[295].CMD := 1; Lines[295].Param := 0; // G1 Linear
    Lines[296].X := 95.101; Lines[296].Z := -148.019; Lines[296].F := 300; Lines[296].CMD := 1; Lines[296].Param := 0; // G1 Linear
    Lines[297].X := 94.284; Lines[297].Z := -148.547; Lines[297].F := 300; Lines[297].CMD := 1; Lines[297].Param := 0; // G1 Linear
    Lines[298].X := 93.436; Lines[298].Z := -149.062; Lines[298].F := 300; Lines[298].CMD := 1; Lines[298].Param := 0; // G1 Linear
    Lines[299].X := 92.558; Lines[299].Z := -149.562; Lines[299].F := 300; Lines[299].CMD := 1; Lines[299].Param := 0; // G1 Linear
    Lines[300].X := 91.652; Lines[300].Z := -150.049; Lines[300].F := 300; Lines[300].CMD := 1; Lines[300].Param := 0; // G1 Linear
    Lines[301].X := 90.719; Lines[301].Z := -150.523; Lines[301].F := 300; Lines[301].CMD := 1; Lines[301].Param := 0; // G1 Linear
    Lines[302].X := 89.761; Lines[302].Z := -150.982; Lines[302].F := 300; Lines[302].CMD := 1; Lines[302].Param := 0; // G1 Linear
    Lines[303].X := 88.780; Lines[303].Z := -151.429; Lines[303].F := 300; Lines[303].CMD := 1; Lines[303].Param := 0; // G1 Linear
    Lines[304].X := 87.777; Lines[304].Z := -151.862; Lines[304].F := 300; Lines[304].CMD := 1; Lines[304].Param := 0; // G1 Linear
    Lines[305].X := 86.754; Lines[305].Z := -152.283; Lines[305].F := 300; Lines[305].CMD := 1; Lines[305].Param := 0; // G1 Linear
    Lines[306].X := 85.712; Lines[306].Z := -152.690; Lines[306].F := 300; Lines[306].CMD := 1; Lines[306].Param := 0; // G1 Linear
    Lines[307].X := 84.654; Lines[307].Z := -153.085; Lines[307].F := 300; Lines[307].CMD := 1; Lines[307].Param := 0; // G1 Linear
    Lines[308].X := 83.580; Lines[308].Z := -153.467; Lines[308].F := 300; Lines[308].CMD := 1; Lines[308].Param := 0; // G1 Linear
    Lines[309].X := 82.493; Lines[309].Z := -153.836; Lines[309].F := 300; Lines[309].CMD := 1; Lines[309].Param := 0; // G1 Linear
    Lines[310].X := 81.393; Lines[310].Z := -154.193; Lines[310].F := 300; Lines[310].CMD := 1; Lines[310].Param := 0; // G1 Linear
    Lines[311].X := 80.284; Lines[311].Z := -154.538; Lines[311].F := 300; Lines[311].CMD := 1; Lines[311].Param := 0; // G1 Linear
    Lines[312].X := 79.165; Lines[312].Z := -154.871; Lines[312].F := 300; Lines[312].CMD := 1; Lines[312].Param := 0; // G1 Linear
    Lines[313].X := 78.040; Lines[313].Z := -155.192; Lines[313].F := 300; Lines[313].CMD := 1; Lines[313].Param := 0; // G1 Linear
    Lines[314].X := 76.909; Lines[314].Z := -155.501; Lines[314].F := 300; Lines[314].CMD := 1; Lines[314].Param := 0; // G1 Linear
    Lines[315].X := 75.775; Lines[315].Z := -155.798; Lines[315].F := 300; Lines[315].CMD := 1; Lines[315].Param := 0; // G1 Linear
    Lines[316].X := 74.638; Lines[316].Z := -156.084; Lines[316].F := 300; Lines[316].CMD := 1; Lines[316].Param := 0; // G1 Linear
    Lines[317].X := 73.501; Lines[317].Z := -156.358; Lines[317].F := 300; Lines[317].CMD := 1; Lines[317].Param := 0; // G1 Linear
    Lines[318].X := 72.364; Lines[318].Z := -156.621; Lines[318].F := 300; Lines[318].CMD := 1; Lines[318].Param := 0; // G1 Linear
    Lines[319].X := 71.231; Lines[319].Z := -156.873; Lines[319].F := 300; Lines[319].CMD := 1; Lines[319].Param := 0; // G1 Linear
    Lines[320].X := 70.102; Lines[320].Z := -157.114; Lines[320].F := 300; Lines[320].CMD := 1; Lines[320].Param := 0; // G1 Linear
    Lines[321].X := 68.979; Lines[321].Z := -157.344; Lines[321].F := 300; Lines[321].CMD := 1; Lines[321].Param := 0; // G1 Linear
    Lines[322].X := 67.863; Lines[322].Z := -157.564; Lines[322].F := 300; Lines[322].CMD := 1; Lines[322].Param := 0; // G1 Linear
    Lines[323].X := 66.757; Lines[323].Z := -157.772; Lines[323].F := 300; Lines[323].CMD := 1; Lines[323].Param := 0; // G1 Linear
    Lines[324].X := 65.662; Lines[324].Z := -157.971; Lines[324].F := 300; Lines[324].CMD := 1; Lines[324].Param := 0; // G1 Linear
    Lines[325].X := 64.579; Lines[325].Z := -158.159; Lines[325].F := 300; Lines[325].CMD := 1; Lines[325].Param := 0; // G1 Linear
    Lines[326].X := 63.511; Lines[326].Z := -158.337; Lines[326].F := 300; Lines[326].CMD := 1; Lines[326].Param := 0; // G1 Linear
    Lines[327].X := 62.458; Lines[327].Z := -158.504; Lines[327].F := 300; Lines[327].CMD := 1; Lines[327].Param := 0; // G1 Linear
    Lines[328].X := 61.422; Lines[328].Z := -158.662; Lines[328].F := 300; Lines[328].CMD := 1; Lines[328].Param := 0; // G1 Linear
    Lines[329].X := 60.406; Lines[329].Z := -158.810; Lines[329].F := 300; Lines[329].CMD := 1; Lines[329].Param := 0; // G1 Linear
    Lines[330].X := 40.406; Lines[330].Z := -138.810; Lines[330].F := 0; Lines[330].CMD := 0; Lines[330].Param := 0; // G0 Rapid
    Lines[331].X := 80.252; Lines[331].Z := -118.936; Lines[331].F := 0; Lines[331].CMD := 0; Lines[331].Param := 0; // G0 Rapid
    Lines[332].X := 81.079; Lines[332].Z := -119.545; Lines[332].F := 300; Lines[332].CMD := 1; Lines[332].Param := 0; // G1 Linear
    Lines[333].X := 81.920; Lines[333].Z := -120.173; Lines[333].F := 300; Lines[333].CMD := 1; Lines[333].Param := 0; // G1 Linear
    Lines[334].X := 82.773; Lines[334].Z := -120.818; Lines[334].F := 300; Lines[334].CMD := 1; Lines[334].Param := 0; // G1 Linear
    Lines[335].X := 83.637; Lines[335].Z := -121.481; Lines[335].F := 300; Lines[335].CMD := 1; Lines[335].Param := 0; // G1 Linear
    Lines[336].X := 84.512; Lines[336].Z := -122.160; Lines[336].F := 300; Lines[336].CMD := 1; Lines[336].Param := 0; // G1 Linear
    Lines[337].X := 85.396; Lines[337].Z := -122.855; Lines[337].F := 300; Lines[337].CMD := 1; Lines[337].Param := 0; // G1 Linear
    Lines[338].X := 86.288; Lines[338].Z := -123.566; Lines[338].F := 300; Lines[338].CMD := 1; Lines[338].Param := 0; // G1 Linear
    Lines[339].X := 87.187; Lines[339].Z := -124.291; Lines[339].F := 300; Lines[339].CMD := 1; Lines[339].Param := 0; // G1 Linear
    Lines[340].X := 88.092; Lines[340].Z := -125.031; Lines[340].F := 300; Lines[340].CMD := 1; Lines[340].Param := 0; // G1 Linear
    Lines[341].X := 89.002; Lines[341].Z := -125.785; Lines[341].F := 300; Lines[341].CMD := 1; Lines[341].Param := 0; // G1 Linear
    Lines[342].X := 89.917; Lines[342].Z := -126.552; Lines[342].F := 300; Lines[342].CMD := 1; Lines[342].Param := 0; // G1 Linear
    Lines[343].X := 90.834; Lines[343].Z := -127.332; Lines[343].F := 300; Lines[343].CMD := 1; Lines[343].Param := 0; // G1 Linear
    Lines[344].X := 91.753; Lines[344].Z := -128.124; Lines[344].F := 300; Lines[344].CMD := 1; Lines[344].Param := 0; // G1 Linear
    Lines[345].X := 92.674; Lines[345].Z := -128.928; Lines[345].F := 300; Lines[345].CMD := 1; Lines[345].Param := 0; // G1 Linear
    Lines[346].X := 93.594; Lines[346].Z := -129.743; Lines[346].F := 300; Lines[346].CMD := 1; Lines[346].Param := 0; // G1 Linear
    Lines[347].X := 94.512; Lines[347].Z := -130.568; Lines[347].F := 300; Lines[347].CMD := 1; Lines[347].Param := 0; // G1 Linear
    Lines[348].X := 95.429; Lines[348].Z := -131.404; Lines[348].F := 300; Lines[348].CMD := 1; Lines[348].Param := 0; // G1 Linear
    Lines[349].X := 96.342; Lines[349].Z := -132.249; Lines[349].F := 300; Lines[349].CMD := 1; Lines[349].Param := 0; // G1 Linear
    Lines[350].X := 97.251; Lines[350].Z := -133.103; Lines[350].F := 300; Lines[350].CMD := 1; Lines[350].Param := 0; // G1 Linear
    Lines[351].X := 98.155; Lines[351].Z := -133.965; Lines[351].F := 300; Lines[351].CMD := 1; Lines[351].Param := 0; // G1 Linear
    Lines[352].X := 99.052; Lines[352].Z := -134.835; Lines[352].F := 300; Lines[352].CMD := 1; Lines[352].Param := 0; // G1 Linear
    Lines[353].X := 99.942; Lines[353].Z := -135.713; Lines[353].F := 300; Lines[353].CMD := 1; Lines[353].Param := 0; // G1 Linear
    Lines[354].X := 100.824; Lines[354].Z := -136.597; Lines[354].F := 300; Lines[354].CMD := 1; Lines[354].Param := 0; // G1 Linear
    Lines[355].X := 101.695; Lines[355].Z := -137.488; Lines[355].F := 300; Lines[355].CMD := 1; Lines[355].Param := 0; // G1 Linear
    Lines[356].X := 102.557; Lines[356].Z := -138.384; Lines[356].F := 300; Lines[356].CMD := 1; Lines[356].Param := 0; // G1 Linear
    Lines[357].X := 103.406; Lines[357].Z := -139.285; Lines[357].F := 300; Lines[357].CMD := 1; Lines[357].Param := 0; // G1 Linear
    Lines[358].X := 104.244; Lines[358].Z := -140.191; Lines[358].F := 300; Lines[358].CMD := 1; Lines[358].Param := 0; // G1 Linear
    Lines[359].X := 105.067; Lines[359].Z := -141.101; Lines[359].F := 300; Lines[359].CMD := 1; Lines[359].Param := 0; // G1 Linear
    Lines[360].X := 105.876; Lines[360].Z := -142.014; Lines[360].F := 300; Lines[360].CMD := 1; Lines[360].Param := 0; // G1 Linear
    Lines[361].X := 106.669; Lines[361].Z := -142.931; Lines[361].F := 300; Lines[361].CMD := 1; Lines[361].Param := 0; // G1 Linear
    Lines[362].X := 107.445; Lines[362].Z := -143.849; Lines[362].F := 300; Lines[362].CMD := 1; Lines[362].Param := 0; // G1 Linear
    Lines[363].X := 108.203; Lines[363].Z := -144.770; Lines[363].F := 300; Lines[363].CMD := 1; Lines[363].Param := 0; // G1 Linear
    Lines[364].X := 108.943; Lines[364].Z := -145.692; Lines[364].F := 300; Lines[364].CMD := 1; Lines[364].Param := 0; // G1 Linear
    Lines[365].X := 109.662; Lines[365].Z := -146.614; Lines[365].F := 300; Lines[365].CMD := 1; Lines[365].Param := 0; // G1 Linear
    Lines[366].X := 110.361; Lines[366].Z := -147.537; Lines[366].F := 300; Lines[366].CMD := 1; Lines[366].Param := 0; // G1 Linear
    Lines[367].X := 111.037; Lines[367].Z := -148.460; Lines[367].F := 300; Lines[367].CMD := 1; Lines[367].Param := 0; // G1 Linear
    Lines[368].X := 111.691; Lines[368].Z := -149.381; Lines[368].F := 300; Lines[368].CMD := 1; Lines[368].Param := 0; // G1 Linear
    Lines[369].X := 112.320; Lines[369].Z := -150.301; Lines[369].F := 300; Lines[369].CMD := 1; Lines[369].Param := 0; // G1 Linear
    Lines[370].X := 112.924; Lines[370].Z := -151.220; Lines[370].F := 300; Lines[370].CMD := 1; Lines[370].Param := 0; // G1 Linear
    Lines[371].X := 113.502; Lines[371].Z := -152.135; Lines[371].F := 300; Lines[371].CMD := 1; Lines[371].Param := 0; // G1 Linear
    Lines[372].X := 114.053; Lines[372].Z := -153.048; Lines[372].F := 300; Lines[372].CMD := 1; Lines[372].Param := 0; // G1 Linear
    Lines[373].X := 114.576; Lines[373].Z := -153.957; Lines[373].F := 300; Lines[373].CMD := 1; Lines[373].Param := 0; // G1 Linear
    Lines[374].X := 115.069; Lines[374].Z := -154.862; Lines[374].F := 300; Lines[374].CMD := 1; Lines[374].Param := 0; // G1 Linear
    Lines[375].X := 115.533; Lines[375].Z := -155.762; Lines[375].F := 300; Lines[375].CMD := 1; Lines[375].Param := 0; // G1 Linear
    Lines[376].X := 115.964; Lines[376].Z := -156.657; Lines[376].F := 300; Lines[376].CMD := 1; Lines[376].Param := 0; // G1 Linear
    Lines[377].X := 116.363; Lines[377].Z := -157.546; Lines[377].F := 300; Lines[377].CMD := 1; Lines[377].Param := 0; // G1 Linear
    Lines[378].X := 116.729; Lines[378].Z := -158.428; Lines[378].F := 300; Lines[378].CMD := 1; Lines[378].Param := 0; // G1 Linear
    Lines[379].X := 117.061; Lines[379].Z := -159.304; Lines[379].F := 300; Lines[379].CMD := 1; Lines[379].Param := 0; // G1 Linear
    Lines[380].X := 117.356; Lines[380].Z := -160.173; Lines[380].F := 300; Lines[380].CMD := 1; Lines[380].Param := 0; // G1 Linear
    Lines[381].X := 117.616; Lines[381].Z := -161.033; Lines[381].F := 300; Lines[381].CMD := 1; Lines[381].Param := 0; // G1 Linear
    Lines[382].X := 117.837; Lines[382].Z := -161.885; Lines[382].F := 300; Lines[382].CMD := 1; Lines[382].Param := 0; // G1 Linear
    Lines[383].X := 118.020; Lines[383].Z := -162.728; Lines[383].F := 300; Lines[383].CMD := 1; Lines[383].Param := 0; // G1 Linear
    Lines[384].X := 118.164; Lines[384].Z := -163.561; Lines[384].F := 300; Lines[384].CMD := 1; Lines[384].Param := 0; // G1 Linear
    Lines[385].X := 118.266; Lines[385].Z := -164.384; Lines[385].F := 300; Lines[385].CMD := 1; Lines[385].Param := 0; // G1 Linear
    Lines[386].X := 118.327; Lines[386].Z := -165.196; Lines[386].F := 300; Lines[386].CMD := 1; Lines[386].Param := 0; // G1 Linear
    Lines[387].X := 118.345; Lines[387].Z := -165.997; Lines[387].F := 300; Lines[387].CMD := 1; Lines[387].Param := 0; // G1 Linear
    Lines[388].X := 118.319; Lines[388].Z := -166.786; Lines[388].F := 300; Lines[388].CMD := 1; Lines[388].Param := 0; // G1 Linear
    Lines[389].X := 118.248; Lines[389].Z := -167.563; Lines[389].F := 300; Lines[389].CMD := 1; Lines[389].Param := 0; // G1 Linear
    Lines[390].X := 118.131; Lines[390].Z := -168.327; Lines[390].F := 300; Lines[390].CMD := 1; Lines[390].Param := 0; // G1 Linear
    Lines[391].X := 117.967; Lines[391].Z := -169.078; Lines[391].F := 300; Lines[391].CMD := 1; Lines[391].Param := 0; // G1 Linear
    Lines[392].X := 117.756; Lines[392].Z := -169.814; Lines[392].F := 300; Lines[392].CMD := 1; Lines[392].Param := 0; // G1 Linear
    Lines[393].X := 117.495; Lines[393].Z := -170.536; Lines[393].F := 300; Lines[393].CMD := 1; Lines[393].Param := 0; // G1 Linear
    Lines[394].X := 117.184; Lines[394].Z := -171.243; Lines[394].F := 300; Lines[394].CMD := 1; Lines[394].Param := 0; // G1 Linear
    Lines[395].X := 116.822; Lines[395].Z := -171.935; Lines[395].F := 300; Lines[395].CMD := 1; Lines[395].Param := 0; // G1 Linear
    Lines[396].X := 116.411; Lines[396].Z := -172.610; Lines[396].F := 300; Lines[396].CMD := 1; Lines[396].Param := 0; // G1 Linear
    Lines[397].X := 115.952; Lines[397].Z := -173.271; Lines[397].F := 300; Lines[397].CMD := 1; Lines[397].Param := 0; // G1 Linear
    Lines[398].X := 115.447; Lines[398].Z := -173.916; Lines[398].F := 300; Lines[398].CMD := 1; Lines[398].Param := 0; // G1 Linear
    Lines[399].X := 114.897; Lines[399].Z := -174.547; Lines[399].F := 300; Lines[399].CMD := 1; Lines[399].Param := 0; // G1 Linear
    Lines[400].X := 114.304; Lines[400].Z := -175.162; Lines[400].F := 300; Lines[400].CMD := 1; Lines[400].Param := 0; // G1 Linear
    Lines[401].X := 113.670; Lines[401].Z := -175.762; Lines[401].F := 300; Lines[401].CMD := 1; Lines[401].Param := 0; // G1 Linear
    Lines[402].X := 112.996; Lines[402].Z := -176.348; Lines[402].F := 300; Lines[402].CMD := 1; Lines[402].Param := 0; // G1 Linear
    Lines[403].X := 112.284; Lines[403].Z := -176.919; Lines[403].F := 300; Lines[403].CMD := 1; Lines[403].Param := 0; // G1 Linear
    Lines[404].X := 111.536; Lines[404].Z := -177.476; Lines[404].F := 300; Lines[404].CMD := 1; Lines[404].Param := 0; // G1 Linear
    Lines[405].X := 110.752; Lines[405].Z := -178.019; Lines[405].F := 300; Lines[405].CMD := 1; Lines[405].Param := 0; // G1 Linear
    Lines[406].X := 109.936; Lines[406].Z := -178.547; Lines[406].F := 300; Lines[406].CMD := 1; Lines[406].Param := 0; // G1 Linear
    Lines[407].X := 109.088; Lines[407].Z := -179.062; Lines[407].F := 300; Lines[407].CMD := 1; Lines[407].Param := 0; // G1 Linear
    Lines[408].X := 108.210; Lines[408].Z := -179.562; Lines[408].F := 300; Lines[408].CMD := 1; Lines[408].Param := 0; // G1 Linear
    Lines[409].X := 107.304; Lines[409].Z := -180.049; Lines[409].F := 300; Lines[409].CMD := 1; Lines[409].Param := 0; // G1 Linear
    Lines[410].X := 106.371; Lines[410].Z := -180.523; Lines[410].F := 300; Lines[410].CMD := 1; Lines[410].Param := 0; // G1 Linear
    Lines[411].X := 105.413; Lines[411].Z := -180.982; Lines[411].F := 300; Lines[411].CMD := 1; Lines[411].Param := 0; // G1 Linear
    Lines[412].X := 104.432; Lines[412].Z := -181.429; Lines[412].F := 300; Lines[412].CMD := 1; Lines[412].Param := 0; // G1 Linear
    Lines[413].X := 103.429; Lines[413].Z := -181.862; Lines[413].F := 300; Lines[413].CMD := 1; Lines[413].Param := 0; // G1 Linear
    Lines[414].X := 102.405; Lines[414].Z := -182.283; Lines[414].F := 300; Lines[414].CMD := 1; Lines[414].Param := 0; // G1 Linear
    Lines[415].X := 101.364; Lines[415].Z := -182.690; Lines[415].F := 300; Lines[415].CMD := 1; Lines[415].Param := 0; // G1 Linear
    Lines[416].X := 100.305; Lines[416].Z := -183.085; Lines[416].F := 300; Lines[416].CMD := 1; Lines[416].Param := 0; // G1 Linear
    Lines[417].X := 99.232; Lines[417].Z := -183.467; Lines[417].F := 300; Lines[417].CMD := 1; Lines[417].Param := 0; // G1 Linear
    Lines[418].X := 98.144; Lines[418].Z := -183.836; Lines[418].F := 300; Lines[418].CMD := 1; Lines[418].Param := 0; // G1 Linear
    Lines[419].X := 97.045; Lines[419].Z := -184.193; Lines[419].F := 300; Lines[419].CMD := 1; Lines[419].Param := 0; // G1 Linear
    Lines[420].X := 95.935; Lines[420].Z := -184.538; Lines[420].F := 300; Lines[420].CMD := 1; Lines[420].Param := 0; // G1 Linear
    Lines[421].X := 94.817; Lines[421].Z := -184.871; Lines[421].F := 300; Lines[421].CMD := 1; Lines[421].Param := 0; // G1 Linear
    Lines[422].X := 93.692; Lines[422].Z := -185.192; Lines[422].F := 300; Lines[422].CMD := 1; Lines[422].Param := 0; // G1 Linear
    Lines[423].X := 92.561; Lines[423].Z := -185.501; Lines[423].F := 300; Lines[423].CMD := 1; Lines[423].Param := 0; // G1 Linear
    Lines[424].X := 91.426; Lines[424].Z := -185.798; Lines[424].F := 300; Lines[424].CMD := 1; Lines[424].Param := 0; // G1 Linear
    Lines[425].X := 90.290; Lines[425].Z := -186.084; Lines[425].F := 300; Lines[425].CMD := 1; Lines[425].Param := 0; // G1 Linear
    Lines[426].X := 89.152; Lines[426].Z := -186.358; Lines[426].F := 300; Lines[426].CMD := 1; Lines[426].Param := 0; // G1 Linear
    Lines[427].X := 88.016; Lines[427].Z := -186.621; Lines[427].F := 300; Lines[427].CMD := 1; Lines[427].Param := 0; // G1 Linear
    Lines[428].X := 86.883; Lines[428].Z := -186.873; Lines[428].F := 300; Lines[428].CMD := 1; Lines[428].Param := 0; // G1 Linear
    Lines[429].X := 85.754; Lines[429].Z := -187.114; Lines[429].F := 300; Lines[429].CMD := 1; Lines[429].Param := 0; // G1 Linear
    Lines[430].X := 84.631; Lines[430].Z := -187.344; Lines[430].F := 300; Lines[430].CMD := 1; Lines[430].Param := 0; // G1 Linear
    Lines[431].X := 83.515; Lines[431].Z := -187.564; Lines[431].F := 300; Lines[431].CMD := 1; Lines[431].Param := 0; // G1 Linear
    Lines[432].X := 82.409; Lines[432].Z := -187.772; Lines[432].F := 300; Lines[432].CMD := 1; Lines[432].Param := 0; // G1 Linear
    Lines[433].X := 81.314; Lines[433].Z := -187.971; Lines[433].F := 300; Lines[433].CMD := 1; Lines[433].Param := 0; // G1 Linear
    Lines[434].X := 80.231; Lines[434].Z := -188.159; Lines[434].F := 300; Lines[434].CMD := 1; Lines[434].Param := 0; // G1 Linear
    Lines[435].X := 79.162; Lines[435].Z := -188.337; Lines[435].F := 300; Lines[435].CMD := 1; Lines[435].Param := 0; // G1 Linear
    Lines[436].X := 78.109; Lines[436].Z := -188.504; Lines[436].F := 300; Lines[436].CMD := 1; Lines[436].Param := 0; // G1 Linear
    Lines[437].X := 77.074; Lines[437].Z := -188.662; Lines[437].F := 300; Lines[437].CMD := 1; Lines[437].Param := 0; // G1 Linear
    Lines[438].X := 76.058; Lines[438].Z := -188.810; Lines[438].F := 300; Lines[438].CMD := 1; Lines[438].Param := 0; // G1 Linear
    Lines[439].X := 56.058; Lines[439].Z := -168.810; Lines[439].F := 0; Lines[439].CMD := 0; Lines[439].Param := 0; // G0 Rapid
    Lines[440].X := 0.000; Lines[440].Z := -168.810; Lines[440].F := 0; Lines[440].CMD := 0; Lines[440].Param := 0; // G0 Rapid
    Lines[441].X := 0.000; Lines[441].Z := 0.000; Lines[441].F := 0; Lines[441].CMD := 0; Lines[441].Param := 0; // G0 Rapid
    Lines[442].X := 0.000; Lines[442].Z := 0.000; Lines[442].F := 0; Lines[442].CMD := 21; Lines[442].Param := 0; // Spindle OFF
    Lines[443].X := 0.000; Lines[443].Z := 0.000; Lines[443].F := 0; Lines[443].CMD := 21; Lines[443].Param := 0; // Spindle OFF
    Lines[444].X := 0.000; Lines[444].Z := 0.000; Lines[444].F := 0; Lines[444].CMD := 99; Lines[444].Param := 0; // Program END
END_DATA_BLOCK